# EPICS substitutions: elioApp/Db/EL4104.substitutions
file EL4104.template { pattern
{ CHAN	}
{ 1	}
{ 2	}
{ 3	}
{ 4	}
}
